RoboDK station: ProyectoFINAL_OYOLA_HERRERA.rdk

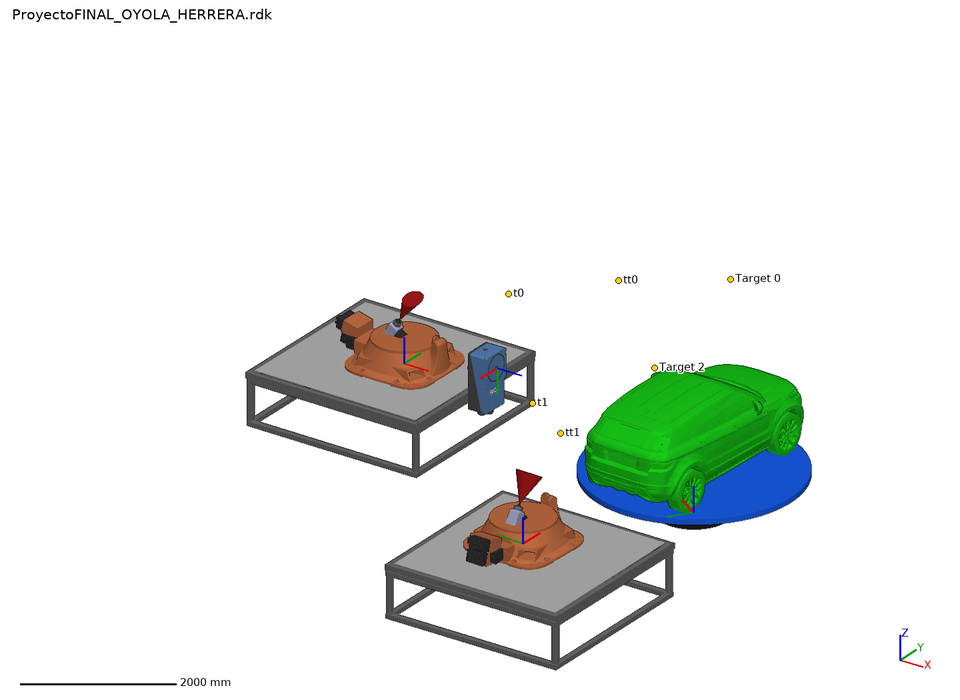
[picture v0: the station drawn from its stored meshes, robots at their saved joint values, targets as dots, program paths as lines]
Station ProyectoFINAL_OYOLA_HERRERA (saved by RoboDK 5.2.4). Poses are relative to the parent item; angles as X-Y-Z fixed-axis rotations.
Station parameters (name, value as stored): ColorAuto, Verde, SENSOR, 1, correo, majorp1993@gmail.com
  - frame Mesa_Juguete at (810, -1300, 250.84) mm, rotated rx 0 ry 0 rz 148.51 deg
    - robot Eje Externo: 1 axes
        modified DH rows (alpha deg, a mm, theta deg, d mm): 0, 0, 0, 0
        joint limits [0] to [360]; home [0]; saved at [360]
      - object Eje Externo Base at (0, 0, 0) mm, size 2999.6 x 2999.8 x 625 mm
      - object RangeOver at (0, 0, 0) mm, rotated rx 0 ry 0 rz 30 deg, size 1721.2 x 1253 x 3335.7 mm, geometry from range over.obj
    - target Target 0 (joint target) at (-235.79, -405.13, 3335.88) mm, rotated rx 176.34 ry 31.8 rz -61.18 deg; joints [-6.222, -56.523, 13.833, 3.485, 70.875, -6.426, 0] of KUKA KR 1000 titan
  - frame ROBOTO at (600, -4800, 1144.75) mm, rotated rx 0 ry 0 rz 88.43 deg
    - robot KUKA KR 1000 titan: 6 axes, payload 1000 kg, reach 3202 mm, repeatability 0.2 mm, weight 4690 kg
        joint limits [-150, -130, -110, -350, -118, -350] to [150, 17.5, 145, 350, 118, 350]; home [0, -90, 90, 0, 0, 0]; saved at [22.341, -98.53, 95.267, -12.974, 63.826, 25.019]
      - tool Paint gun, TCP at (100, 0, 900) mm, rotated rx 0 ry 30 rz 0 deg, size 406.4 x 559.5 x 943.1 mm
    - object Table 108x114x32 IN at (1219.03, -129.11, -820.76) mm, rotated rx 0 ry 0 rz -178.23 deg, size 2628.9 x 2679.7 x 778.4 mm, geometry from Table-108x114x32-IN.sld
    - target t0 (Cartesian target) at (235.79, 405.13, 3335.88) mm, rotated rx 176.34 ry 31.8 rz 118.82 deg; joints [-6.222, -56.523, 13.833, 3.485, 70.875, -6.426, 0] of KUKA KR 1000 titan
    - target t1 (Cartesian target) at (357.2, 117.73, 1814.4) mm, rotated rx 180 ry 2 rz 119.93 deg; joints [-84.253, -48.412, -86.816, 161.152, 106.957, 25.645, 0] of KUKA KR 1000 titan
  - frame ROBOTN at (-3560, -1500, 1219.08) mm
    - robot KUKA KR 1000 titan2 (model KUKA KR 1000 titan): 6 axes, payload 1000 kg, reach 3202 mm, repeatability 0.2 mm, weight 4690 kg
        joint limits [-150, -130, -110, -350, -118, -350] to [150, 17.5, 145, 350, 118, 350]; home [0, -90, 90, 0, 0, 0]; saved at [-10.198, -63.866, 102.536, -7.017, -57.322, 4.648]
      - tool Paint gunN, TCP at (100, 0, 500) mm, rotated rx 0 ry 17 rz 0 deg, size 406.4 x 559.5 x 943.1 mm
    - object Table 108x114x32 IN at (-208.03, -1343.21, -782.6) mm, rotated rx 0 ry -0.09 rz 89.8 deg, size 2628.9 x 2679.7 x 778.4 mm, geometry from Table-108x114x32-IN.sld
    - target Target 2 (Cartesian target) at (3307.48, 849.02, 518.46) mm, rotated rx 180 ry 89.15 rz 180 deg; joints [-22.42, -13.743, 94.046, -21.667, -97.158, 3.712] of KUKA KR 1000 titan2
    - target tt0 (Cartesian target) at (3016.44, 450.03, 1837.55) mm, rotated rx 38.03 ry 88.27 rz 42.35 deg; joints [-10.198, -63.866, 102.536, -7.017, -57.322, 4.648] of KUKA KR 1000 titan2
    - target tt1 (Cartesian target) at (3248.68, -1170.53, 387.77) mm, rotated rx 38.04 ry 88.27 rz 42.35 deg; joints [27.254, -3.671, 61.537, 29.931, -80.502, -17.358] of KUKA KR 1000 titan2
    - frame framecamera at (1450, 0, 340) mm, rotated rx -90 ry 0 rz -90 deg
      - object SICK VSPP-5f2113 at (0, 0, -280) mm, rotated rx 0 ry 0 rz -90 deg, size 424 x 928 x 304 mm, geometry from Cam2D_SICK_VSPP_5F2113.sld
  - Python program parametros (listed below)
  - Python program SprayOn (listed below)
  - Python program EnviaCorreo (listed below)
  - Python program TomarFoto (listed below)
  - Python program PrepareSimulation (listed below)
  - Python program 0TechoConP (listed below)
  - Python program 0LateralConP (listed below)
  - Python program 180LateralConP (listed below)
  - Python program 180CapotConP (listed below)
  - Python program 270LateralConP (listed below)
  - program ALLMOVE (10 instructions, listed below)
  - program TomaFotoYenvia (2 instructions, listed below)

--- Python program parametros ---
from robolink import *    # RoboDK API
from robodk import *      # Robot toolbox
RDK = Robolink()

#Variables Globales
PARAM_COLOR_AUTO='ColorAuto'
PARAM_CORREO_DESTINO = 'correo'
PARAM_fin= ''


RDK= Robolink()

color_auto=RDK.getParam(PARAM_COLOR_AUTO)

coloresL=['Blanco','Gris','Negro','Amarillo','Verde']
colores='\n1)Blanco\n2)Gris\n3)Negro\n4)Amarillo\n5)Verde'

coloresCod=[[1,1,1],[0.5,0.5,0.5],[0.15,0.15,0.15],[0.85,0.85,0],[0,0.85,0]]

Ncolor_input= mbox('Ingrese el numero de color que desea que se pinte el carro'+str(colores), entry='1')

color_input= coloresCod[int(Ncolor_input)-1]
color_nombre= coloresL[int(Ncolor_input)-1]

RDK.setParam(PARAM_COLOR_AUTO, color_nombre)

#parametro de foto antes o despues
RDK.setParam(PARAM_fin,0)


correo_input= mbox('Ingrese el correo al cual desea enviar las fotos', entry='jaoyola99@gmail.com')
RDK.setParam(PARAM_CORREO_DESTINO,correo_input)

--- Python program SprayOn ---
# This macro allows simulating a spray gun
# It is possible to call SprayOn(1) to simulate turning the Spray gun ON or GunOn(0) to stop simulating the gun
# Calling SprayOn(-1) clears all displayed data
# The macro will output spray gun statistics

# For more information visit:
# http://www.robodk.com/doc/PythonAPI/robolink.html

# Define the default action (0 to deactivate, +1 to activate, -1 to clear any spray gun simulation)
# Setting it to None will display a message
ACTION = 1

from robolink import *    # API to communicate with RoboDK
from robodk import *      # basic matrix operations
RDK = Robolink()

# quit if we are not in simulation mode
if RDK.RunMode() != RUNMODE_SIMULATE:
    quit()

# Get any previously added spray gun simulations and display statistics (spray on the part vs spray falling out of the part)
info, data = RDK.Spray_GetStats()
if data.size(1) > 0:
    print("Spray gun statistics:")
    print(info)
    print(data.tr())
    # # Diplay statistics
    # RDK.ShowMessage("Material used: %.1f%%<br>Material waisted: %.1f%%<br>Total particles: %.1f" % (data[1,0],data[2,0],data[3,0]), True)
    # # Clear previous spray
    # RDK.Spray_Clear()

# Check if we are running this program inside another program and passing arguments
import sys
if len(sys.argv) > 1:
    ACTION = int(sys.argv[1])

# If the default ACTION is None, display a message to activate/deactivate the spray gun
if ACTION is None:
    print('Note: This macro can be called as GunOn(1) or GunOn(0)')
    entry = mbox('Turn gun ON or OFF', ('On', '1'), ('Off', '0'))
    if not entry:
        quit()
    ACTION = int(entry)

if ACTION == 0:
    # Turn the gun off
    RDK.Spray_SetState(SPRAY_OFF)

if ACTION < 0:
    # Clear all spray simulations
    RDK.Spray_Clear()

elif ACTION > 0:
    # Create a new spray gun object in RoboDK
    # by using RDK.Spray_Add(tool, object, options_command, volume, geometry)
    # tool: tool item (TCP) to use
    # object: object to project the particles
    # options_command (optional): string to specify options. Example:
    #     STEP=AxB: Defines the grid to be projected 1x1 means only one line of particle projection (for example, for welding)
    #     PARTICLE: Defines the shape and size of particle (sphere or particle), unless a specific geometry is provided:
    #       a- SPHERE(radius, facets)
    #       b- SPHERE(radius, facets, scalex, scaley, scalez)
    #       b- CUBE(sizex, sizey, sizez)
    #     RAND=factor: Defines a random factor factor 0 means that the particles are not deposited randomly
    #     ELLYPSE: defines the volume as an ellypse (default)
    #     RECTANGLE: defines the volume as a rectangle
    #     PROJECT: project the particles to the surface (default) (for welding, painting or scanning)
    #     NO_PROJECT: does not project the particles to the surface (for example, for 3D printing)
    #
    # volume (optional): Matrix of parameters defining the volume of the spray gun
    # geometry (optional): Matrix of vertices defining the triangles.


    tool = 0    # auto detect active tool
    obj = 0     # auto detect object in active reference frame
    # We can specify a given tool object and/or object
    #robot = RDK.Item("ABB IRB 2600-12/1.85", ITEM_TYPE_ROBOT)
    #tools = robot.Childs()
    #if len(tools) > 0:
    #    tool = tools[0]
    #obj = RDK.Item('object', ITEM_TYPE_OBJECT)

    options_command = "ELLYPSE PROJECT PARTICLE=SPHERE(4,8,1,1,0.5) STEP=8x8 RAND=2" # simulate
    #options_command = "PARTICLE=CUBE(10,10,2) STEP=8x8"
    #options_command = "PARTICLE=SPHERE(4,8) STEP=8x8"
    #options_command = "PARTICLE=SPHERE(4,8,1,1,0.1) STEP=8x8 RAND=3"

    # Example commands for welding:
    # options_command = "PROJECT PARTICLE=SPHERE(4,8)"
    # options_command = PARTICLE=SPHERE(4,8) STEP=1x0


    # define the ellypse volume as p0, pA, pB, colorRGBA (close and far), in mm
    # coordinates must be provided with respect to the TCP
    close_p0 = [   0,   0, -200] # xyz in mm
    close_pA = [   5,   0, -200] # xyz in mm
    close_pB = [   0,  10, -200] # xyz in mm
    close_color = [ 1, 0, 0, 1]  # RGBA (0-1)

    far_p0   = [   0,   0,  50] # xyz in mm
    far_pA   = [  60,   0,  50] # xyz in mm
    far_pB   = [   0, 120,  50] # xyz in mm
    far_color   = [ 0, 0, 1, 0.2]  # RGBA (0-1)

    close_param = close_p0 + close_pA + close_pB + close_color
    far_param = far_p0 + far_pA + far_pB + far_color
    volume = Mat([close_param, far_param]).tr()
    RDK.Spray_Add(tool, obj, options_command, volume)
    RDK.Spray_SetState(SPRAY_ON)


    # Another example with a varying rectancular shape
    # define the rectangular volume as p0, pA, pB, colorRGBA (close and far)
    # close_param = [-90,-117,  0,  90,-117,0,   -90,117,  0,       0.2,0.2,1,.1]
    # far_param   = [-175,-190,200, 175,-190,200,   -175,190,200,   0.5,0,0,.9]
    # volume = Mat([close_param, far_param])
    # RDK.Spray_Add(tool, obj, "RECTANGLE PARTICLE=SPHERE(2,5) STEP=15x15 RAND=3", volume.tr())
    # RDK.Spray_SetState(SPRAY_ON)

    # Optional: define geometry as a list of triangles with normals (instead of a scaled cube or a sphere)
    # geom = Mat([[0,0,0,   0,0,1], [5,0,0,   0,0,1], [0,5,0,   0,0,1]])
    # RDK.Spray_Add(tool, obj, "STEP=8x8 RANDX=3", volume.tr(), geom.tr())
    # RDK.Spray_SetState(SPRAY_ON)

--- Python program EnviaCorreo ---
# Importamos librerías
import smtplib
import mimetypes
from robolink import *                                  # import the robolink library (bridge with RoboDK)


# Importamos los módulos necesarios
from email.mime.multipart import MIMEMultipart
from email.mime.image import MIMEImage
from email.encoders import encode_base64

#Variable Global para saber si ya termino de pintar
RDK = Robolink()
PARAM_CORREO_DESTINO = 'correo'
PARAM_fin= ''
termino=RDK.getParam(PARAM_fin)
termino=int(termino)
print(termino)

#configuramos el Destinatario
destino=RDK.getParam(PARAM_CORREO_DESTINO)
#destino= "jaoyola99@gmail.com"

# Creamos objeto Multipart, quien será el recipiente que enviaremos
msg = MIMEMultipart()
msg['From']="josedelgado2540@gmail.com"
msg['To']= destino
msg['Subject']="Correo con imagen Adjunta"

# Adjuntamos Imagen
path_rdk = RDK.getParam("PATH_OPENSTATION")
file_name=path_rdk+'/foto.jpg'
file = open(file_name, "rb")
attach_image = MIMEImage(file.read())

if(termino==1):
    attach_image.add_header('Content-Disposition', 'attachment; filename = "Foto Despues.png"')
else:
    attach_image.add_header('Content-Disposition', 'attachment; filename = "Foto Antes.png"')
msg.attach(attach_image)

# Autenticamos
mailServer = smtplib.SMTP('smtp.gmail.com',587)             #Servidor smtp de google con su puerto
mailServer.ehlo()
mailServer.starttls()
mailServer.ehlo()
mailServer.login("josedelgado2540@gmail.com","Jose1234")

# Enviamos
mailServer.sendmail("josedelgado2540@gmail.com", destino , msg.as_string())

# Cerramos conexión
mailServer.close()

--- Python program TomarFoto ---
from robolink import *    # RoboDK API
from robodk import *      # Robot toolbox
RDK = Robolink()

SENSOR_VARIABLE = "SENSOR"
RDK.setParam(SENSOR_VARIABLE, 1)

path_rdk = RDK.getParam("PATH_OPENSTATION")
file_name = "/foto.jpg" #"RoboDK-Screenshot-HQ" + date_str + ".png"

#RDK.Render(False)
fotos=1
while(fotos>0):
    ref_cam = RDK.Item("framecamera",ITEM_TYPE_FRAME)
    #print(ref_cam)
    ref_cam.setVisible(False)
    #ref_cam.setPose(RDK.ViewPose()) #.inv()*rotx(pi))
    #print(RDK.ViewPose())
    #RDk.Render(True)

    cam_id = RDK.Cam2D_Add(ref_cam, 'FOCAL_LENGHT=6 FOV=60 FAR_LENGHT=2500 SIZE=920x640 BG_COLOR=black')


    #ventana para ajustes de camara
    #cam_id = RDK.Cam2D_Add(ref_cam, 'POPUP')

    #img = cv2.imread(path_rdk+file_name,0)
    def WaitSensor():
        if RDK.RunMode() == RUNMODE_SIMULATE:
            while RDK.getParam(SENSOR_VARIABLE) == 0:
                pause(0.001)
        else:
                RDK.RunProgram('WaitSensor')
        print("part detected")

    WaitSensor()

    RDK.Cam2D_Snapshot((path_rdk+file_name), cam_id)
    print(path_rdk+file_name)
    RDK.Cam2D_Close(cam_id)

    #ref_cam.Delete()
    cam_id.Delete()
    print("Done")
    #RDK.ShowMessage("Foto guardada: " + file_path, False)


    fotos-=1

--- Python program PrepareSimulation ---
from robolink import *    # RoboDK API
from robodk import *      # Robot toolbox
from random import choice
RDK = Robolink()

#Llamamos al robot para ponerlo en su pos inicial
robot = RDK.Item('KUKA KR 1000 titan', ITEM_TYPE_ROBOT)      # retrieve the robot by name
t0Techo = RDK.Item('Target 0', ITEM_TYPE_TARGET)                   #home

robot.MoveJ(t0Techo)



PARAM_COLOR_AUTO='ColorAuto'
PARAM_CORREO_DESTINO = 'CorreoDestino'

#_________Colores al azar_________
coloresCod=[[1,1,1],[0.75,0.75,0.75],[0.15,0.15,0.15],[0.30,0.30,0],[0.8,0,0.40],[0,0.92,0.75],[0.5,1,0.83],[1,0.71,0.76],[0.82,0.41,0.12],[0.29,0,0.51],[0.72,0.53,0.04]]

carro=RDK.Item('RangeOver')


carro.Recolor(choice(coloresCod))
#-_-_-_-_-_-_-_-_-_-_-_-_-_-_-_-_-

--- Python program 0TechoConP ---
from robolink import *                                  # import the robolink library (bridge with RoboDK)
from robodk import *                                    # basic matrix operations


RDK = Robolink()                                        # establish a link with the simulator
robot = RDK.Item('KUKA KR 1000 titan', ITEM_TYPE_ROBOT)      # retrieve the robot by name


frame_r = RDK.Item('ROBOTO', ITEM_TYPE_FRAME)

frame_mc = RDK.Item('Mesa_Juguete', ITEM_TYPE_FRAME)
robot.setPoseFrame(frame_r)



#robot.setJoints([10.43, -63.5, 50.34, -5.78, 71.66, 10.69,0])

t0Techo = RDK.Item('t0', ITEM_TYPE_TARGET)               #home
t1Techo = RDK.Item('t1', ITEM_TYPE_TARGET)               #Primer punto del techo

robot.MoveJ(t0Techo)
robot.MoveJ(t1Techo)

#robot.setPoseFrame(frame_r)                        #cambia el sistema de referencia del robot kuka al frame mesa1
#robot.setPoseFrame(frame_mc)

# calculate a new approach position 100 mm along the Z axis of the tool with respect to the target



a1=transl(1400,0,0)                   #xyz  xposi izq           yposi arriba          zposi
a2=transl(0,-250,0)
a3=transl(-1400,0,0)
a4=transl(0,-250,0)
a5=transl(1400,0,0)
a6=transl(0,-250,0)
a7=transl(-1380,0,0)


A=[a1,a2,a3,a4,a5,a6,a7]
approach=t1Techo.Pose()*transl(0,0,0)
print(t1Techo.Pose())
for i in range(len(A)):
    approach = approach*A[i]
    robot.MoveL(approach)               # linear move to the approach position

robot.MoveJ(t0Techo)

--- Python program 0LateralConP ---
from robolink import *                                  # import the robolink library (bridge with RoboDK)
from robodk import *                                    # basic matrix operations



RDK = Robolink()                                        # establish a link with the simulator
robot = RDK.Item('KUKA KR 1000 titan2', ITEM_TYPE_ROBOT)      # retrieve the robot by name
robotO = RDK.Item('KUKA KR 1000 titan', ITEM_TYPE_ROBOT)

frame_r = RDK.Item('ROBOTN', ITEM_TYPE_FRAME)

#2
frame_mc = RDK.Item('Mesa_Juguete', ITEM_TYPE_FRAME)




#robot.setJoints([10.43, -63.5, 50.34, -5.78, 71.66, 10.69,0])

tt0Lateral0 = RDK.Item('tt0', ITEM_TYPE_TARGET)               #home
tt1Lateral1 = RDK.Item('tt1', ITEM_TYPE_TARGET)               #Primer punto del lateral a 0grados
robot.MoveJ(tt0Lateral0)
robot.MoveJ(tt1Lateral1)


# calculate a new approach position 100 mm along the Z axis of the tool with respect to the target

compe1=280           #Compoensacion por q el carro no esta centrado
compe2=180           #Compensacion por la forma del carro
                                    #REFERENCIA con el carro vertical
a1=transl(compe2,2500,compe1)                   #zx  xposi izq           yposi arriba          zposi abajo
a2=transl(150,0,0)                          #baja
a3=transl(-compe2,-2500,-compe1)
a4=transl(250,0,0)
a5=transl(-250,500,50)
a6=transl(200,280,0)
a7=transl(50,1200,130)
a8=transl(180,0,0)
a9=transl(-50,-1200,-130)

A=[a1,a2,a3,a4,a5,a6,a7,a8,a9]
approach=tt1Lateral1.Pose()*transl(0,0,0)
for i in range(len(A)):
    approach = approach*A[i]
    robot.MoveL(approach)               # linear move to the approach position
robot.MoveJ(tt0Lateral0)



#Girar 180 la mesa, 7ma articulacion
joints = robotO.Joints().list()          # retrieve the current robot joints as a list
print(joints)
joints[6] = 180                           # set joint 7 to 0 deg
robotO.MoveJ(joints)                     # move the robot to the new joint position



#RDK.ShowMessage('----Fin----')

--- Python program 180LateralConP ---
from robolink import *                                  # import the robolink library (bridge with RoboDK)
from robodk import *                                    # basic matrix operations



RDK = Robolink()                                        # establish a link with the simulator
robot = RDK.Item('KUKA KR 1000 titan2', ITEM_TYPE_ROBOT)      # retrieve the robot by name
robotO = RDK.Item('KUKA KR 1000 titan', ITEM_TYPE_ROBOT)

frame_r = RDK.Item('ROBOTN', ITEM_TYPE_FRAME)

#2
frame_mc = RDK.Item('Mesa_Juguete', ITEM_TYPE_FRAME)




#robot.setJoints([10.43, -63.5, 50.34, -5.78, 71.66, 10.69,0])

tt0Lateral0 = RDK.Item('tt0', ITEM_TYPE_TARGET)               #home
tt1Lateral1 = RDK.Item('tt1', ITEM_TYPE_TARGET)               #Primer punto del lateral a 0grados

robot.MoveJ(tt0Lateral0)
#robot.MoveJ(tt1Lateral1)


# calculate a new approach position 100 mm along the Z axis of the tool with respect to the target

compe1=320           #Compoensacion por q el carro no esta centrado
compe2=130           #Compensacion por la forma del carro
                                    #REFERENCIA con el carro vertical
a0= transl(460,00,0)                         #Poss inicial lateral 2
#a1= transl(compe2,2500,compe1)                   #zx  xposi izq           yposi arriba          zposi abajo
a1= transl(-300,100,0)
a2= transl(-compe2,2600,compe1)                          #mueve a a izqd
a3= transl(150,0,0)                                      #Baja
a4= transl(compe2,-2000,-compe1)                      #Mueve Dere
a5= transl(100,100,20)                                    #Baja inclinado
a6= transl(0,1120,compe1-180)
a7= transl(180,0,50)
a8= transl(-20,-1140,-200)
a9= transl(0,400,-400)


A=[a0,a1,a2,a3,a4,a5,a6,a7,a8,a9]
approach=tt1Lateral1.Pose()*transl(0,0,0)

for i in range(len(A)):
    approach = approach*A[i]
    robot.MoveL(approach)               # linear move to the approach position

robot.MoveJ(tt0Lateral0)

#Girar 270 la mesa, 7ma articulacion
joints = robotO.Joints().list()          # retrieve the current robot joints as a list
print(joints)
joints[6] = 270                           # set joint 7 to 0 deg
robotO.MoveJ(joints)                     # move the robot to the new joint position

--- Python program 180CapotConP ---
from robolink import *                                  # import the robolink library (bridge with RoboDK)
from robodk import *                                    # basic matrix operations


RDK = Robolink()                                        # establish a link with the simulator
robot = RDK.Item('KUKA KR 1000 titan', ITEM_TYPE_ROBOT)      # retrieve the robot by name


frame_r = RDK.Item('ROBOTO', ITEM_TYPE_FRAME)

frame_mc = RDK.Item('Mesa_Juguete', ITEM_TYPE_FRAME)
robot.setPoseFrame(frame_mc)



#robot.setJoints([10.43, -63.5, 50.34, -5.78, 71.66, 10.69,0])


#robot.MoveJ(t0Techo)


#robot.setPoseFrame(frame_r)                        #cambia el sistema de referencia del robot kuka al frame mesa1
#robot.setPoseFrame(frame_mc)

#Ponemos al inico de donde va a pintar
joints=[-10.71, -67.78, 104.01, 14.66, 22.89, -22.66, 180]
robot.MoveJ(joints)                     # move the robot to the new joint position
#creamos un tarjet con la plataforma girada
        #robot.setPoseFrame(frame_mc)
RDK.AddTarget("T180", frame_mc)
#lo ocultamos
item4=RDK.Item('t180')
item4.setVisible(False)

t0Techo = RDK.Item('T180', ITEM_TYPE_TARGET)               #home


a1=transl(650,0,100)                   #xyz  xposi izq           yposi arriba          zposi baja
a2=transl(0,-250,0)                    #derecha
a3=transl(-550,0,-100)
a4=transl(0,-250,0)
a5=transl(580,0,100)
a6=transl(0,-250,0)
a7=transl(-580,0,-100)
a8=transl(0,-250,0)
a9=transl(500,0,100)
a10=transl(0,0,-1000)

A=[a1,a2,a3,a4,a5,a6,a7,a8,a9,a10]
approach=t0Techo.Pose()*transl(0,0,0)
#borramos el Target
item4.Delete()

for i in range(len(A)):
    approach = approach*A[i]
    robot.MoveL(approach)               # linear move to the approach position

#robot.MoveJ(t0Techo)

--- Python program 270LateralConP ---
from robolink import *                                  # import the robolink library (bridge with RoboDK)
from robodk import *                                    # basic matrix operations


RDK = Robolink()                                        # establish a link with the simulator
robot = RDK.Item('KUKA KR 1000 titan2', ITEM_TYPE_ROBOT)      # retrieve the robot by name
robotO = RDK.Item('KUKA KR 1000 titan', ITEM_TYPE_ROBOT)

frame_r = RDK.Item('ROBOTN', ITEM_TYPE_FRAME)
#2
frame_mc = RDK.Item('Mesa_Juguete', ITEM_TYPE_FRAME)

#Variables Globales
PARAM_COLOR_AUTO='ColorAuto'
PARAM_fin= ''


#robot.setJoints([10.43, -63.5, 50.34, -5.78, 71.66, 10.69,0])

tt0Lateral0 = RDK.Item('tt0', ITEM_TYPE_TARGET)               #home
tt1Lateral1 = RDK.Item('tt1', ITEM_TYPE_TARGET)               #Primer punto del lateral a 0grados

robot.MoveJ(tt0Lateral0)
#robot.MoveJ(tt1Lateral1)


# calculate a new approach position 100 mm along the Z axis of the tool with respect to the target

compe1=320           #Compoensacion por q el carro no esta centrado
compe2=130           #Compensacion por la forma del carro
                                    #REFERENCIA con el carro vertical
a0= transl(0,900,-480)                         #Poss inicial lateral 2
#a1= transl(compe2,2500,compe1)                   #zx  xposi izq           yposi arriba          zposi abajo
a1= transl(0,1100,0)
a3= transl(150,0,0)                                      #Baja
a4= transl(0,-1000,0)                      #Mueve Dere
a5= transl(150,0,0)                                    #Baja
a6= transl(0,900,0)
a7= transl(150,0,-30)



A=[a0,a1,a3,a4,a5,a6,a7,a7]
approach=tt1Lateral1.Pose()*transl(0,0,0)

for i in range(len(A)):
    approach = approach*A[i]
    robot.MoveJ(approach)               # linear move to the approach position

robot.MoveJ(tt0Lateral0)


#Girar 360 la mesa, 7ma articulacion
joints = robotO.Joints().list()          # retrieve the current robot joints as a list
joints[6] = 360                           # set joint 7 to 0 deg
robotO.MoveJ(joints)                     # move the robot to the new joint position



#repitar con el color selecionado
carro=RDK.Item('RangeOver')
color_input=RDK.getParam(PARAM_COLOR_AUTO)
#print(color_input)

colores=['Blanco','Gris','Negro','Amarillo','Verde']

coloresCod=[[1,1,1],[0.5,0.5,0.5],[0.15,0.15,0.15],[0.85,0.85,0],[0,0.85,0]]

a=colores.index(color_input)                #indice

carro.Recolor(coloresCod[a])
#_____________

#enviar senial de q se termino de pintar
RDK.setParam(PARAM_fin,1)



RDK.ShowMessage('El juguete se pinto de color: %s, revise su correo.' %colores[a])

--- program ALLMOVE (robot KUKA KR 1000 titan) ---
  Llamar PrepareSimulation
  Llamar parametros
  Call SprayOn
  Llamar TomaFotoYenvia
  Ejecutar 0TechoConP
  Llamar 0LateralConP
  Ejecutar 180CapotConP
  Llamar 180LateralConP
  Llamar 270LateralConP
  Llamar TomaFotoYenvia

--- program TomaFotoYenvia (robot KUKA KR 1000 titan) ---
  Llamar TomarFoto
  Llamar EnviaCorreo
